FUNCTION_BLOCK LIMIT_ANY (* Abstract superclass for IEC 61131-3 limiters *)
  (* Standard: 61131-3 *)
  (* Version 0.0, 2004-12-15, JHC, Rockwell Automation, Converted from SRC format. *)
  (* Compiler header: package fb.rt.plc.select; *)
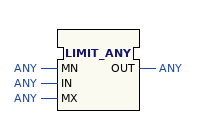
  VAR_INPUT
    MN : ANY; (* Lower limit *)
    IN : ANY; (* Value to be limited *)
    MX : ANY; (* Upper limit *)
  END_VAR
  VAR_OUTPUT
    OUT : ANY; (* MIN(MAX(IN,MN),MX) *)
  END_VAR
END_FUNCTION_BLOCK
